Fanuc KAREL source: wcontaxisvel.kl

PROGRAM wcontaxisvel
%NOLOCKGROUP
VAR
  p : POSITION
  q : POSITION
  i : INTEGER
  r : REAL
BEGIN
  WITH $CONTAXISVEL = 10.0 MOVE TO p
END wcontaxisvel
